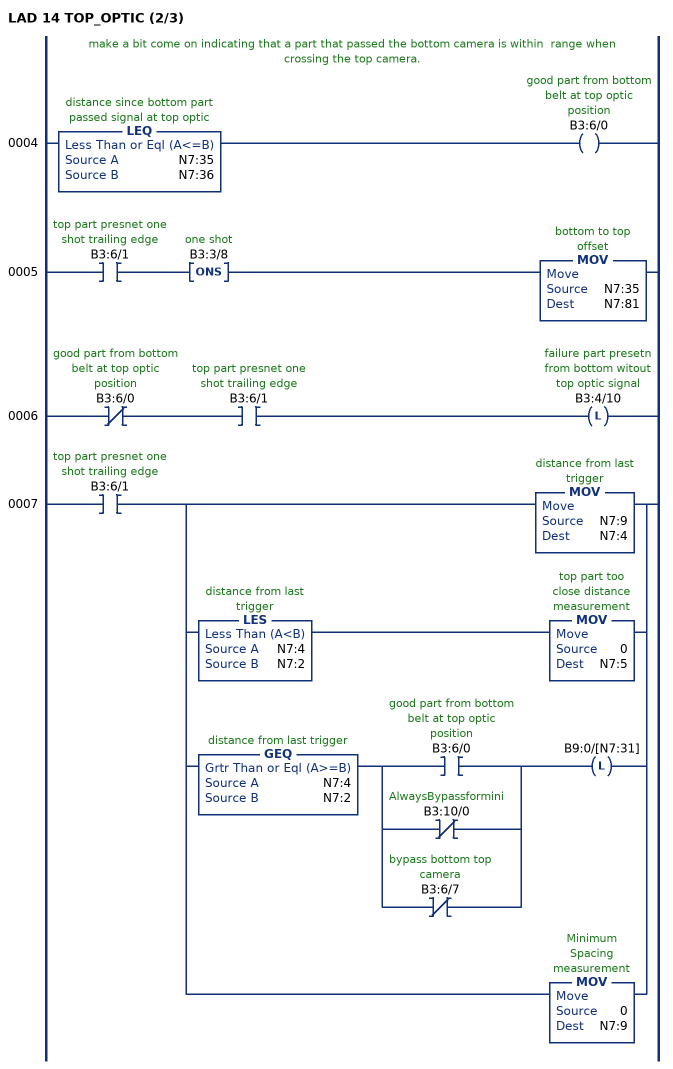
% Rung: 4 %
% make a bit come on indicating that a part that passed the bottom camera is within  range when crossing the top camera. %
SOR LEQ N7:35 N7:36 OTE B3:6/0 EOR
%   N7:35  "distance since bottom part passed signal at top optic" %
%   N7:36  "distance to allow for part shift when part travels from bottom belt to top optic" %
%   B3:6/0  "good part from bottom belt at top optic position" %
% Rung: 5 %
SOR XIC B3:6/1 ONS B3:3/8 MOV N7:35 N7:81 EOR
%   B3:6/1  "top part presnet one shot trailing edge" %
%   B3:3/8  "one shot" %
%   N7:35  "distance since bottom part passed signal at top optic" %
%   N7:81  "bottom to top offset" %
% Rung: 6 %
SOR XIO B3:6/0 XIC B3:6/1 OTL B3:4/10 EOR
%   B3:6/0  "good part from bottom belt at top optic position" %
%   B3:6/1  "top part presnet one shot trailing edge" %
%   B3:4/10  "failure part presetn from bottom witout top optic signal" %
% Rung: 7 %
SOR XIC B3:6/1 BST MOV N7:9 N7:4 NXB LES N7:4 N7:2 MOV 0 N7:5 NXB GEQ N7:4 N7:2 BST XIC B3:6/0 NXB XIO B3:10/0 NXB XIO B3:6/7 BND OTL B9:0/[N7:31] NXB MOV 0 N7:9 BND EOR
%   B3:6/1  "top part presnet one shot trailing edge" %
%   N7:9  "Minimum Spacing measurement" %
%   N7:4  "distance from last trigger" %
%   N7:2  "Min Part Spacing top" %
%   N7:5  "top part too close distance measurement" %
%   B3:6/0  "good part from bottom belt at top optic position" %
%   B3:10/0  "AlwaysBypassformini" %
%   B3:6/7  "bypass bottom top camera" %
%   N7:31  TOP_PART_LOAD_PT %

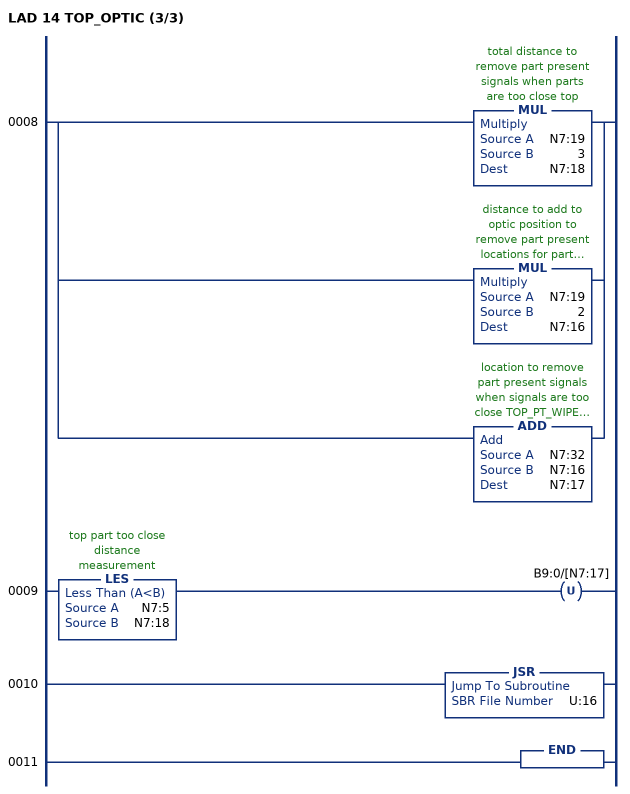
% Rung: 8 %
SOR BST MUL N7:19 3 N7:18 NXB MUL N7:19 2 N7:16 NXB ADD N7:32 N7:16 N7:17 BND EOR
%   N7:19  "distance to remove trigger signals when part spacing too close top" %
%   N7:18  "total distance to remove part present signals when parts are too close top" %
%   N7:16  "distance to add to optic position to remove part present locations for parts too close top" %
%   N7:32  OPTIC_POSITION  "top optic location" %
%   N7:17  TOP_PT_WIPE_LOC  "location to remove part present signals when signals are too close" %
% Rung: 9 %
SOR LES N7:5 N7:18 OTU B9:0/[N7:17] EOR
%   N7:5  "top part too close distance measurement" %
%   N7:18  "total distance to remove part present signals when parts are too close top" %
%   N7:17  TOP_PT_WIPE_LOC  "location to remove part present signals when signals are too close" %
% Rung: 10 %
SOR JSR U:16 EOR
% Rung: 11 %
SOR END EOR

LADDER 16 "TOP_SIDE"
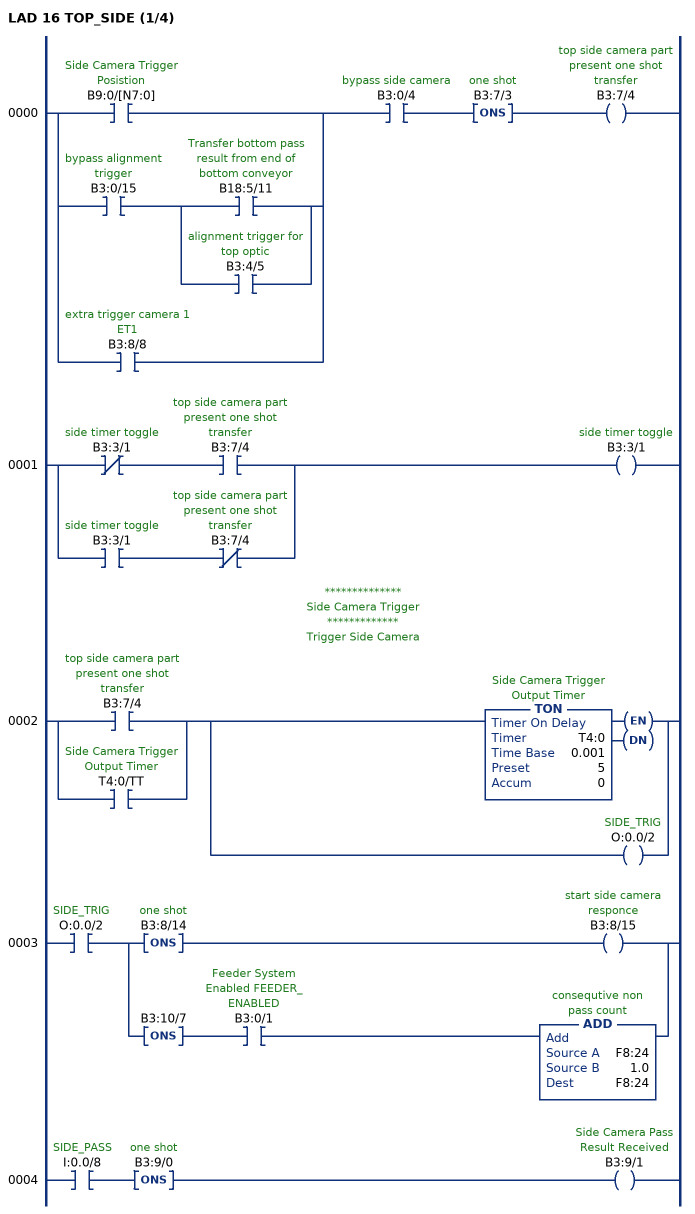
% Rung: 0 %
SOR BST XIC B9:0/[N7:0] NXB XIC B3:0/15 BST XIC B18:5/11 NXB XIC B3:4/5 BND NXB XIC B3:8/8 BND XIC B3:0/4 ONS B3:7/3 OTE B3:7/4 EOR
%   B9:0/[N7:0]  "Side Camera Trigger Posistion" %
%   N7:0  CAMERA_1_SIDE  "Trigger Position" %
%   B3:0/15  "bypass alignment trigger" %
%   B18:5/11  "Transfer bottom pass result from end of bottom conveyor" %
%   B3:4/5  "alignment trigger for top optic" %
%   B3:8/8  ET1  "extra trigger camera 1" %
%   B3:0/4  "bypass side camera" %
%   B3:7/3  "one shot" %
%   B3:7/4  "top side camera part present one shot transfer" %
% Rung: 1 %
SOR BST XIO B3:3/1 XIC B3:7/4 NXB XIC B3:3/1 XIO B3:7/4 BND OTE B3:3/1 EOR
%   B3:3/1  "side timer toggle" %
%   B3:7/4  "top side camera part present one shot transfer" %
% Rung: 2 %
% **************
% Side Camera Trigger
% *************
% 
% Trigger Side Camera %
SOR BST XIC B3:7/4 NXB XIC T4:0/TT BND BST TON T4:0 0.001 5 0 NXB OTE O:0.0/2 BND EOR
%   B3:7/4  "top side camera part present one shot transfer" %
%   T4:0  "Side Camera Trigger Output Timer" %
%   O:0.0/2  SIDE_TRIG %
% Rung: 3 %
SOR XIC O:0.0/2 BST ONS B3:8/14 OTE B3:8/15 NXB ONS B3:10/7 XIC B3:0/1 ADD F8:24 1.0 F8:24 BND EOR
%   O:0.0/2  SIDE_TRIG %
%   B3:8/14  "one shot" %
%   B3:8/15  "start side camera responce" %
%   B3:0/1  FEEDER_ENABLED  "Feeder System Enabled" %
%   F8:24  "consequtive non pass count" %
% Rung: 4 %
SOR XIC I:0.0/8 ONS B3:9/0 OTE B3:9/1 EOR
%   I:0.0/8  SIDE_PASS %
%   B3:9/0  "one shot" %
%   B3:9/1  "Side Camera Pass Result Received" %

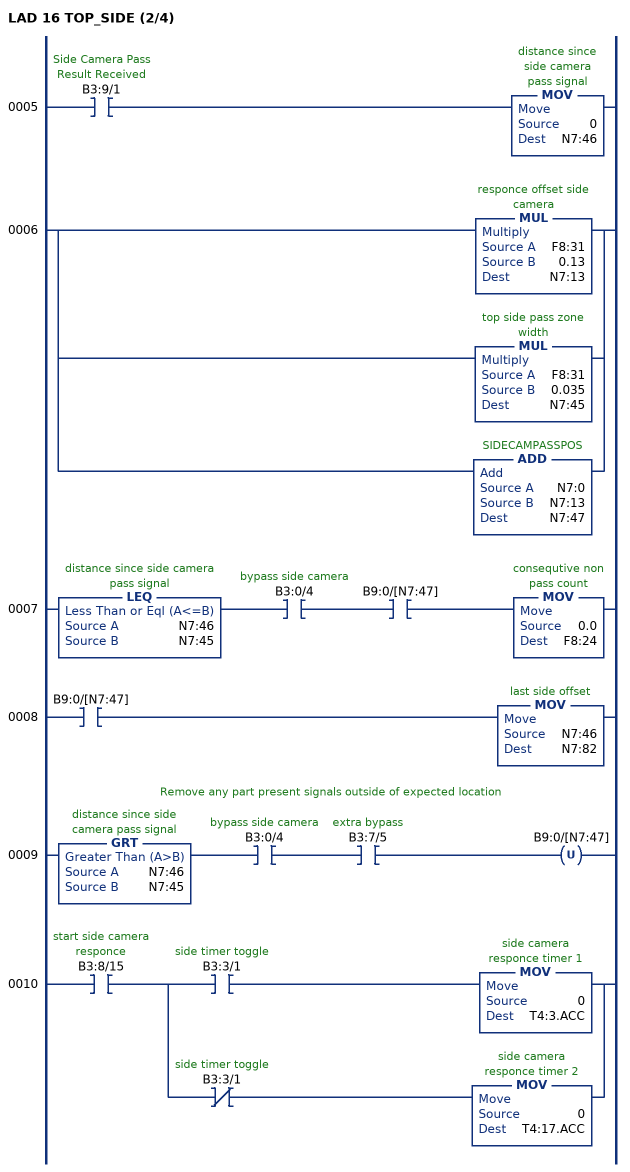
% Rung: 5 %
SOR XIC B3:9/1 MOV 0 N7:46 EOR
%   B3:9/1  "Side Camera Pass Result Received" %
%   N7:46  "distance since side camera pass signal" %
% Rung: 6 %
SOR BST MUL F8:31 0.13 N7:13 NXB MUL F8:31 0.035 N7:45 NXB ADD N7:0 N7:13 N7:47 BND EOR
%   N7:13  "responce offset side camera" %
%   N7:45  "top side pass zone width" %
%   N7:0  CAMERA_1_SIDE  "Trigger Position" %
%   N7:47  SIDECAMPASSPOS %
% Rung: 7 %
SOR LEQ N7:46 N7:45 XIC B3:0/4 XIC B9:0/[N7:47] MOV 0.0 F8:24 EOR
%   N7:46  "distance since side camera pass signal" %
%   N7:45  "top side pass zone width" %
%   B3:0/4  "bypass side camera" %
%   N7:47  SIDECAMPASSPOS %
%   F8:24  "consequtive non pass count" %
% Rung: 8 %
SOR XIC B9:0/[N7:47] MOV N7:46 N7:82 EOR
%   N7:47  SIDECAMPASSPOS %
%   N7:46  "distance since side camera pass signal" %
%   N7:82  "last side offset" %
% Rung: 9 %
% Remove any part present signals outside of expected location %
SOR GRT N7:46 N7:45 XIC B3:0/4 XIC B3:7/5 OTU B9:0/[N7:47] EOR
%   N7:46  "distance since side camera pass signal" %
%   N7:45  "top side pass zone width" %
%   B3:0/4  "bypass side camera" %
%   B3:7/5  "extra bypass" %
%   N7:47  SIDECAMPASSPOS %
% Rung: 10 %
SOR XIC B3:8/15 BST XIC B3:3/1 MOV 0 T4:3.ACC NXB XIO B3:3/1 MOV 0 T4:17.ACC BND EOR
%   B3:8/15  "start side camera responce" %
%   B3:3/1  "side timer toggle" %
%   T4:3  "side camera responce timer 1" %
%   T4:17  "side camera responce timer 2" %

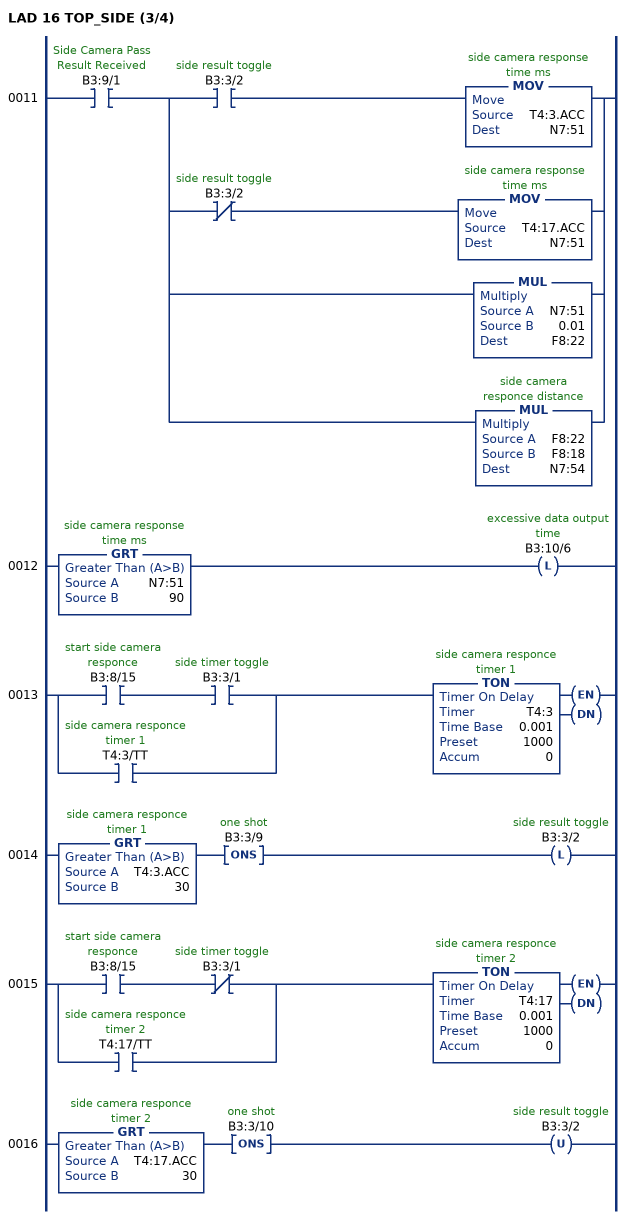
% Rung: 11 %
SOR XIC B3:9/1 BST XIC B3:3/2 MOV T4:3.ACC N7:51 NXB XIO B3:3/2 MOV T4:17.ACC N7:51 NXB MUL N7:51 0.01 F8:22 NXB MUL F8:22 F8:18 N7:54 BND EOR
%   B3:9/1  "Side Camera Pass Result Received" %
%   B3:3/2  "side result toggle" %
%   T4:3  "side camera responce timer 1" %
%   N7:51  "side camera response time ms" %
%   T4:17  "side camera responce timer 2" %
%   F8:18  "top belt speed average in pulses per 100ms" %
%   N7:54  "side camera responce distance" %
% Rung: 12 %
SOR GRT N7:51 90 OTL B3:10/6 EOR
%   N7:51  "side camera response time ms" %
%   B3:10/6  "excessive data output time" %
% Rung: 13 %
SOR BST XIC B3:8/15 XIC B3:3/1 NXB XIC T4:3/TT BND TON T4:3 0.001 1000 0 EOR
%   B3:8/15  "start side camera responce" %
%   B3:3/1  "side timer toggle" %
%   T4:3  "side camera responce timer 1" %
% Rung: 14 %
SOR GRT T4:3.ACC 30 ONS B3:3/9 OTL B3:3/2 EOR
%   T4:3  "side camera responce timer 1" %
%   B3:3/9  "one shot" %
%   B3:3/2  "side result toggle" %
% Rung: 15 %
SOR BST XIC B3:8/15 XIO B3:3/1 NXB XIC T4:17/TT BND TON T4:17 0.001 1000 0 EOR
%   B3:8/15  "start side camera responce" %
%   B3:3/1  "side timer toggle" %
%   T4:17  "side camera responce timer 2" %
% Rung: 16 %
SOR GRT T4:17.ACC 30 ONS B3:3/10 OTU B3:3/2 EOR
%   T4:17  "side camera responce timer 2" %
%   B3:3/10  "one shot" %
%   B3:3/2  "side result toggle" %

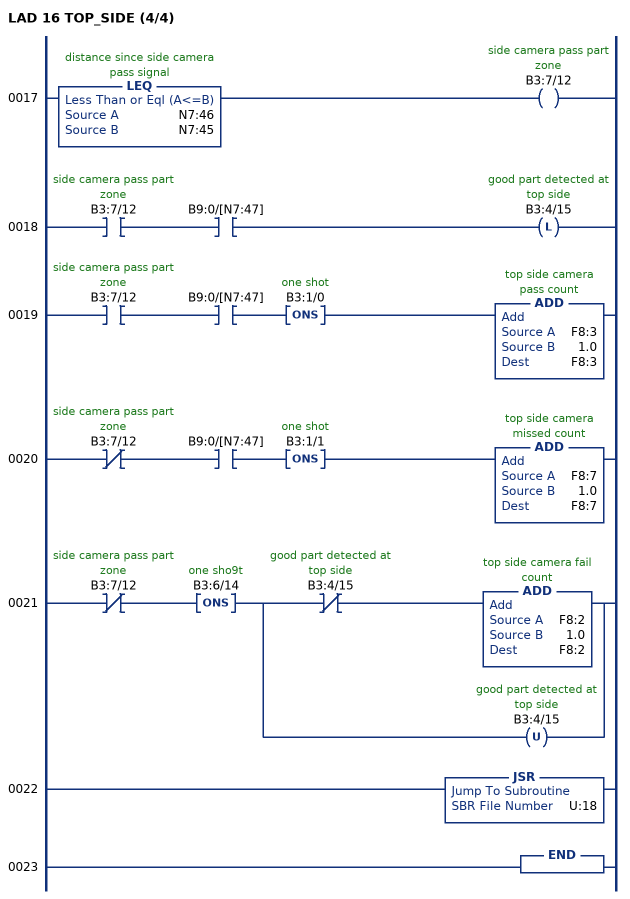
% Rung: 17 %
SOR LEQ N7:46 N7:45 OTE B3:7/12 EOR
%   N7:46  "distance since side camera pass signal" %
%   N7:45  "top side pass zone width" %
%   B3:7/12  "side camera pass part zone" %
% Rung: 18 %
SOR XIC B3:7/12 XIC B9:0/[N7:47] OTL B3:4/15 EOR
%   B3:7/12  "side camera pass part zone" %
%   N7:47  SIDECAMPASSPOS %
%   B3:4/15  "good part detected at top side" %
% Rung: 19 %
SOR XIC B3:7/12 XIC B9:0/[N7:47] ONS B3:1/0 ADD F8:3 1.0 F8:3 EOR
%   B3:7/12  "side camera pass part zone" %
%   N7:47  SIDECAMPASSPOS %
%   B3:1/0  "one shot" %
%   F8:3  "top side camera pass count" %
% Rung: 20 %
SOR XIO B3:7/12 XIC B9:0/[N7:47] ONS B3:1/1 ADD F8:7 1.0 F8:7 EOR
%   B3:7/12  "side camera pass part zone" %
%   N7:47  SIDECAMPASSPOS %
%   B3:1/1  "one shot" %
%   F8:7  "top side camera missed count" %
% Rung: 21 %
SOR XIO B3:7/12 ONS B3:6/14 BST XIO B3:4/15 ADD F8:2 1.0 F8:2 NXB OTU B3:4/15 BND EOR
%   B3:7/12  "side camera pass part zone" %
%   B3:6/14  "one sho9t" %
%   B3:4/15  "good part detected at top side" %
%   F8:2  "top side camera fail count" %
% Rung: 22 %
SOR JSR U:18 EOR
% Rung: 23 %
SOR END EOR

LADDER 18 "TOP_PYRIMI"
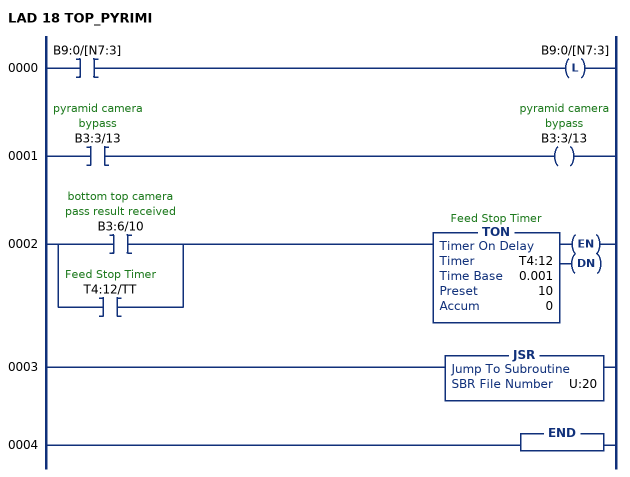
% Rung: 0 %
SOR XIC B9:0/[N7:3] OTL B9:0/[N7:3] EOR
%   N7:3  PYRAMID_TRIG  "pyramid camera trigger position" %
% Rung: 1 %
SOR XIC B3:3/13 OTE B3:3/13 EOR
%   B3:3/13  "pyramid camera bypass" %
% Rung: 2 %
SOR BST XIC B3:6/10 NXB XIC T4:12/TT BND TON T4:12 0.001 10 0 EOR
%   B3:6/10  "bottom top camera pass result received" %
%   T4:12  "Feed Stop Timer" %
% Rung: 3 %
SOR JSR U:20 EOR
% Rung: 4 %
SOR END EOR

LADDER 20 "TOP_TOP"
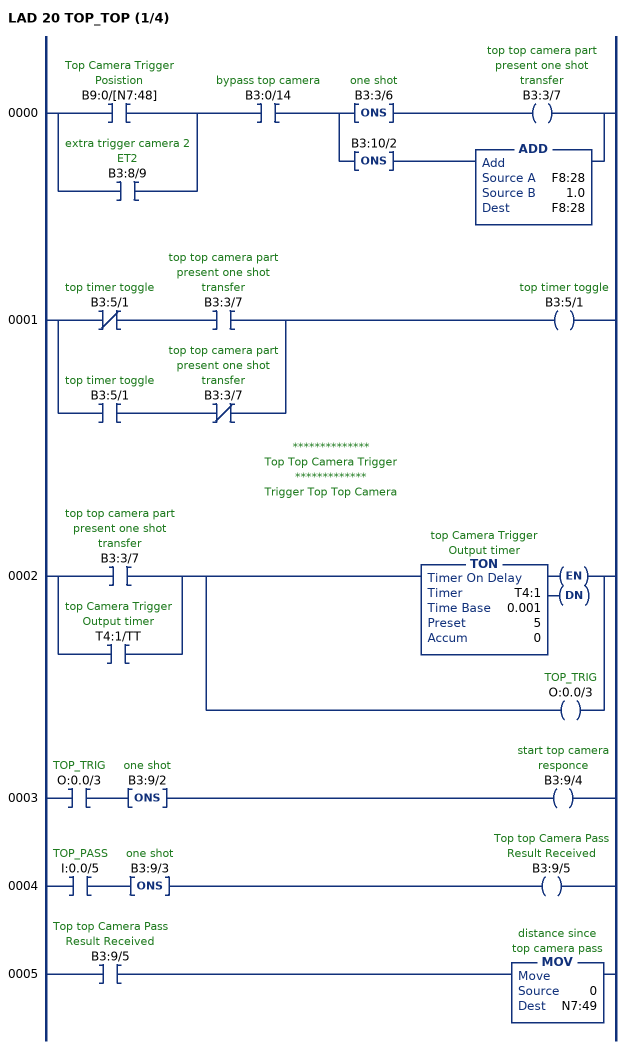
% Rung: 0 %
SOR BST XIC B9:0/[N7:48] NXB XIC B3:8/9 BND XIC B3:0/14 BST ONS B3:3/6 OTE B3:3/7 NXB ONS B3:10/2 ADD F8:28 1.0 F8:28 BND EOR
%   B9:0/[N7:48]  "Top Camera Trigger Posistion" %
%   N7:48  CAMERA_2_TOP  "top camera trigger position" %
%   B3:8/9  ET2  "extra trigger camera 2" %
%   B3:0/14  "bypass top camera" %
%   B3:3/6  "one shot" %
%   B3:3/7  "top top camera part present one shot transfer" %
% Rung: 1 %
SOR BST XIO B3:5/1 XIC B3:3/7 NXB XIC B3:5/1 XIO B3:3/7 BND OTE B3:5/1 EOR
%   B3:5/1  "top timer toggle" %
%   B3:3/7  "top top camera part present one shot transfer" %
% Rung: 2 %
% **************
% Top Top Camera Trigger
% *************
% 
% Trigger Top Top Camera %
SOR BST XIC B3:3/7 NXB XIC T4:1/TT BND BST TON T4:1 0.001 5 0 NXB OTE O:0.0/3 BND EOR
%   B3:3/7  "top top camera part present one shot transfer" %
%   T4:1  "top Camera Trigger Output timer" %
%   O:0.0/3  TOP_TRIG %
% Rung: 3 %
SOR XIC O:0.0/3 ONS B3:9/2 OTE B3:9/4 EOR
%   O:0.0/3  TOP_TRIG %
%   B3:9/2  "one shot" %
%   B3:9/4  "start top camera responce" %
% Rung: 4 %
SOR XIC I:0.0/5 ONS B3:9/3 OTE B3:9/5 EOR
%   I:0.0/5  TOP_PASS %
%   B3:9/3  "one shot" %
%   B3:9/5  "Top top Camera Pass Result Received" %
% Rung: 5 %
SOR XIC B3:9/5 MOV 0 N7:49 EOR
%   B3:9/5  "Top top Camera Pass Result Received" %
%   N7:49  "distance since top camera pass" %

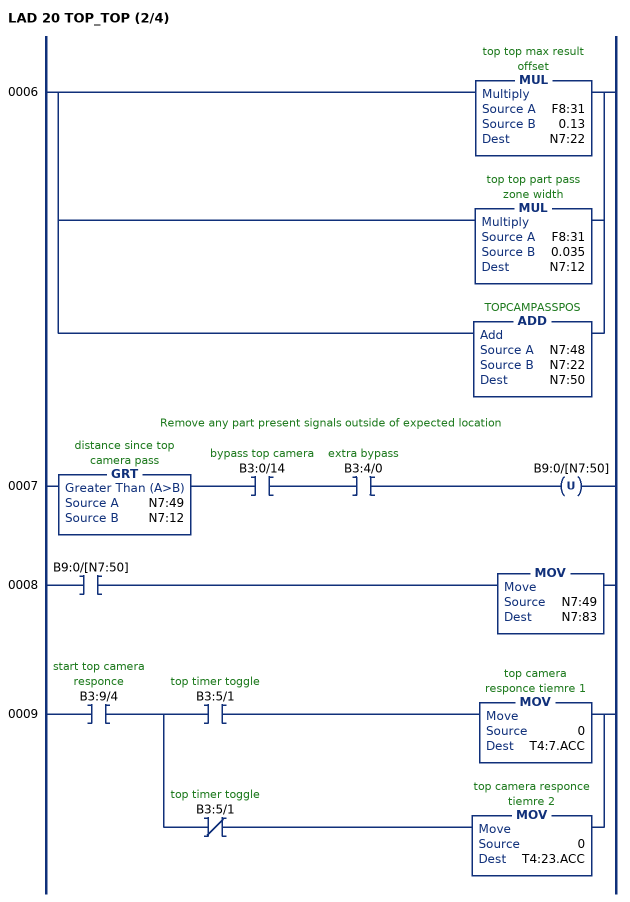
% Rung: 6 %
SOR BST MUL F8:31 0.13 N7:22 NXB MUL F8:31 0.035 N7:12 NXB ADD N7:48 N7:22 N7:50 BND EOR
%   N7:22  "top top max result offset" %
%   N7:12  "top top part pass zone width" %
%   N7:48  CAMERA_2_TOP  "top camera trigger position" %
%   N7:50  TOPCAMPASSPOS %
% Rung: 7 %
% Remove any part present signals outside of expected location %
SOR GRT N7:49 N7:12 XIC B3:0/14 XIC B3:4/0 OTU B9:0/[N7:50] EOR
%   N7:49  "distance since top camera pass" %
%   N7:12  "top top part pass zone width" %
%   B3:0/14  "bypass top camera" %
%   B3:4/0  "extra bypass" %
%   N7:50  TOPCAMPASSPOS %
% Rung: 8 %
SOR XIC B9:0/[N7:50] MOV N7:49 N7:83 EOR
%   N7:50  TOPCAMPASSPOS %
%   N7:49  "distance since top camera pass" %
% Rung: 9 %
SOR XIC B3:9/4 BST XIC B3:5/1 MOV 0 T4:7.ACC NXB XIO B3:5/1 MOV 0 T4:23.ACC BND EOR
%   B3:9/4  "start top camera responce" %
%   B3:5/1  "top timer toggle" %
%   T4:7  "top camera responce tiemre 1" %
%   T4:23  "top camera responce tiemre 2" %

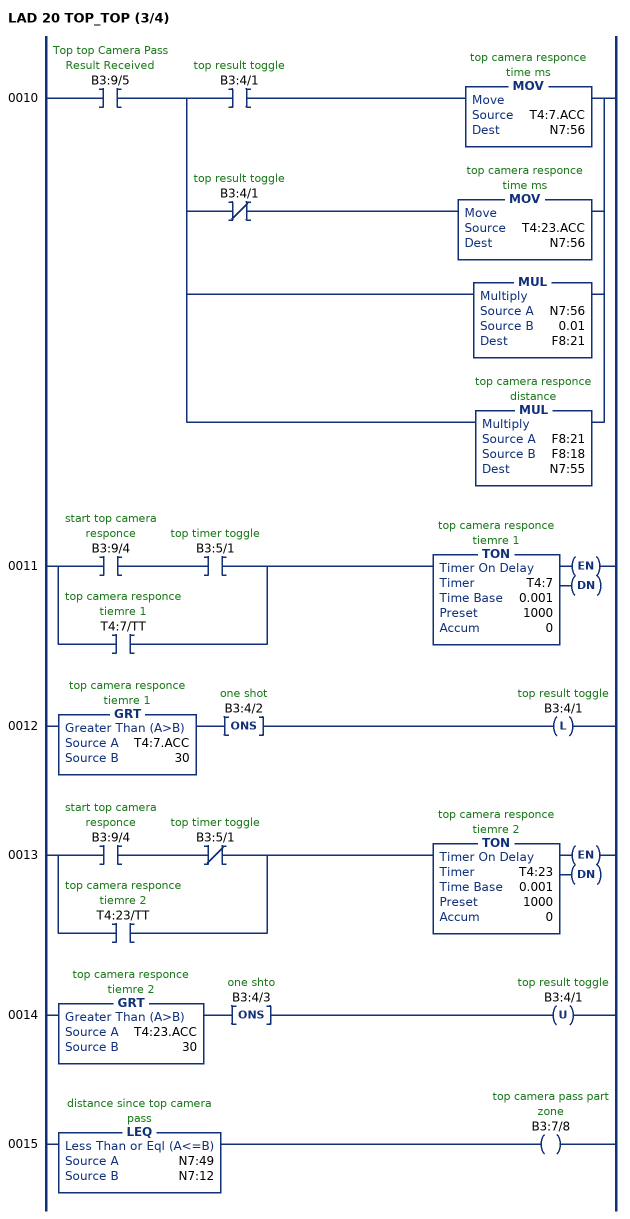
% Rung: 10 %
SOR XIC B3:9/5 BST XIC B3:4/1 MOV T4:7.ACC N7:56 NXB XIO B3:4/1 MOV T4:23.ACC N7:56 NXB MUL N7:56 0.01 F8:21 NXB MUL F8:21 F8:18 N7:55 BND EOR
%   B3:9/5  "Top top Camera Pass Result Received" %
%   B3:4/1  "top result toggle" %
%   T4:7  "top camera responce tiemre 1" %
%   N7:56  "top camera responce time ms" %
%   T4:23  "top camera responce tiemre 2" %
%   F8:18  "top belt speed average in pulses per 100ms" %
%   N7:55  "top camera responce distance" %
% Rung: 11 %
SOR BST XIC B3:9/4 XIC B3:5/1 NXB XIC T4:7/TT BND TON T4:7 0.001 1000 0 EOR
%   B3:9/4  "start top camera responce" %
%   B3:5/1  "top timer toggle" %
%   T4:7  "top camera responce tiemre 1" %
% Rung: 12 %
SOR GRT T4:7.ACC 30 ONS B3:4/2 OTL B3:4/1 EOR
%   T4:7  "top camera responce tiemre 1" %
%   B3:4/2  "one shot" %
%   B3:4/1  "top result toggle" %
% Rung: 13 %
SOR BST XIC B3:9/4 XIO B3:5/1 NXB XIC T4:23/TT BND TON T4:23 0.001 1000 0 EOR
%   B3:9/4  "start top camera responce" %
%   B3:5/1  "top timer toggle" %
%   T4:23  "top camera responce tiemre 2" %
% Rung: 14 %
SOR GRT T4:23.ACC 30 ONS B3:4/3 OTU B3:4/1 EOR
%   T4:23  "top camera responce tiemre 2" %
%   B3:4/3  "one shto" %
%   B3:4/1  "top result toggle" %
% Rung: 15 %
SOR LEQ N7:49 N7:12 OTE B3:7/8 EOR
%   N7:49  "distance since top camera pass" %
%   N7:12  "top top part pass zone width" %
%   B3:7/8  "top camera pass part zone" %

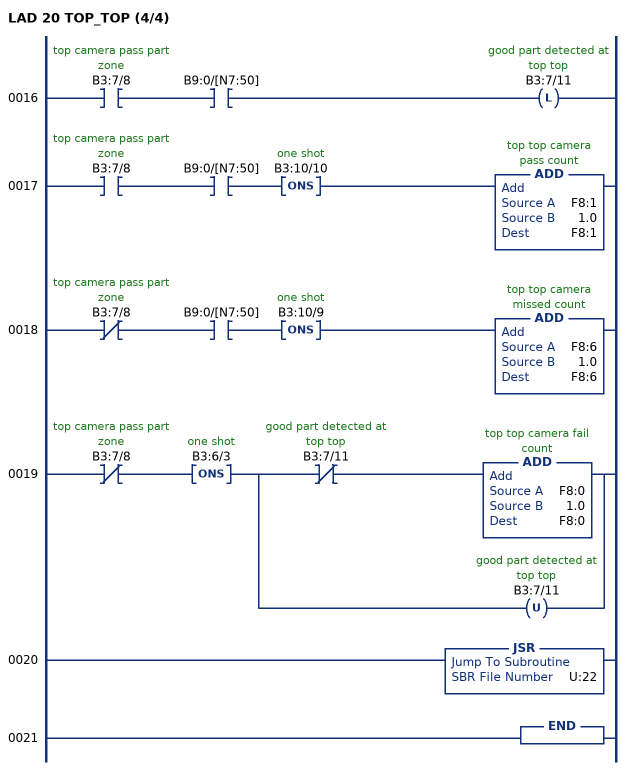
% Rung: 16 %
SOR XIC B3:7/8 XIC B9:0/[N7:50] OTL B3:7/11 EOR
%   B3:7/8  "top camera pass part zone" %
%   N7:50  TOPCAMPASSPOS %
%   B3:7/11  "good part detected at top top" %
% Rung: 17 %
SOR XIC B3:7/8 XIC B9:0/[N7:50] ONS B3:10/10 ADD F8:1 1.0 F8:1 EOR
%   B3:7/8  "top camera pass part zone" %
%   N7:50  TOPCAMPASSPOS %
%   B3:10/10  "one shot" %
%   F8:1  "top top camera pass count" %
% Rung: 18 %
SOR XIO B3:7/8 XIC B9:0/[N7:50] ONS B3:10/9 ADD F8:6 1.0 F8:6 EOR
%   B3:7/8  "top camera pass part zone" %
%   N7:50  TOPCAMPASSPOS %
%   B3:10/9  "one shot" %
%   F8:6  "top top camera missed count" %
% Rung: 19 %
SOR XIO B3:7/8 ONS B3:6/3 BST XIO B3:7/11 ADD F8:0 1.0 F8:0 NXB OTU B3:7/11 BND EOR
%   B3:7/8  "top camera pass part zone" %
%   B3:6/3  "one shot" %
%   B3:7/11  "good part detected at top top" %
%   F8:0  "top top camera fail count" %
% Rung: 20 %
SOR JSR U:22 EOR
% Rung: 21 %
SOR END EOR

LADDER 22 "TOP_THREAD"
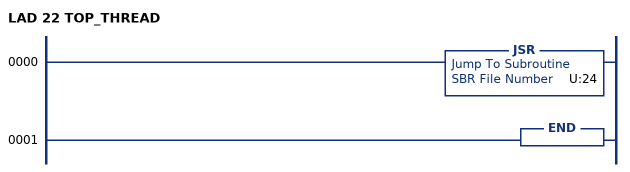
% Rung: 0 %
SOR JSR U:24 EOR
% Rung: 1 %
SOR END EOR

LADDER 24 "TOP_BLOW"
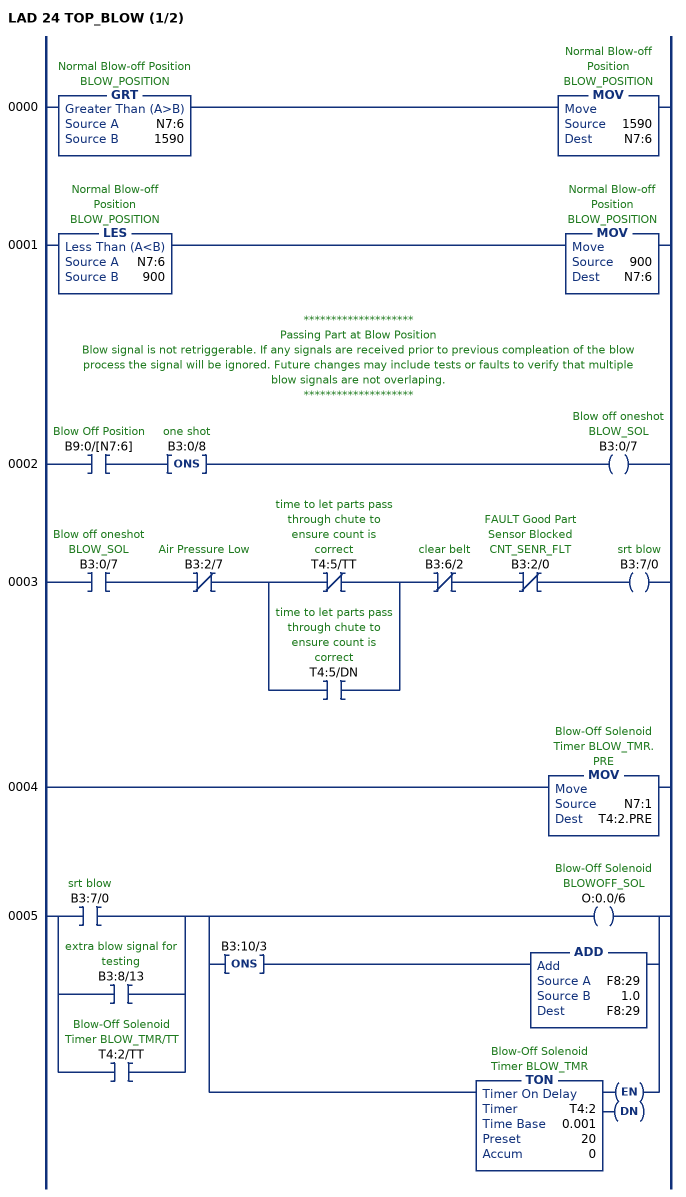
% Rung: 0 %
SOR GRT N7:6 1590 MOV 1590 N7:6 EOR
%   N7:6  BLOW_POSITION  "Normal Blow-off Position" %
% Rung: 1 %
SOR LES N7:6 900 MOV 900 N7:6 EOR
%   N7:6  BLOW_POSITION  "Normal Blow-off Position" %
% Rung: 2 %
% ********************
% Passing Part at Blow Position
% 
% Blow signal is not retriggerable. If any signals are received prior to previous compleation of the blow process the signal will be ignored. Future changes may include tests or faults to verify that multiple blow signals are not overlaping.
% ******************** %
SOR XIC B9:0/[N7:6] ONS B3:0/8 OTE B3:0/7 EOR
%   B9:0/[N7:6]  "Blow Off Position" %
%   N7:6  BLOW_POSITION  "Normal Blow-off Position" %
%   B3:0/8  "one shot" %
%   B3:0/7  BLOW_SOL  "Blow off oneshot" %
% Rung: 3 %
SOR XIC B3:0/7 XIO B3:2/7 BST XIO T4:5/TT NXB XIC T4:5/DN BND XIO B3:6/2 XIO B3:2/0 OTE B3:7/0 EOR
%   B3:0/7  BLOW_SOL  "Blow off oneshot" %
%   B3:2/7  "Air Pressure Low" %
%   T4:5  "time to let parts pass through chute to ensure count is correct" %
%   B3:6/2  "clear belt" %
%   B3:2/0  CNT_SENR_FLT  "FAULT Good Part Sensor Blocked" %
%   B3:7/0  "srt blow" %
% Rung: 4 %
SOR MOV N7:1 T4:2.PRE EOR
%   N7:1  "Blow off Time" %
%   T4:2  BLOW_TMR  "Blow-Off Solenoid Timer" %
% Rung: 5 %
SOR BST XIC B3:7/0 NXB XIC B3:8/13 NXB XIC T4:2/TT BND BST OTE O:0.0/6 NXB ONS B3:10/3 ADD F8:29 1.0 F8:29 NXB TON T4:2 0.001 20 0 BND EOR
%   B3:7/0  "srt blow" %
%   B3:8/13  "extra blow signal for testing" %
%   T4:2  BLOW_TMR  "Blow-Off Solenoid Timer" %
%   O:0.0/6  BLOWOFF_SOL  "Blow-Off Solenoid" %

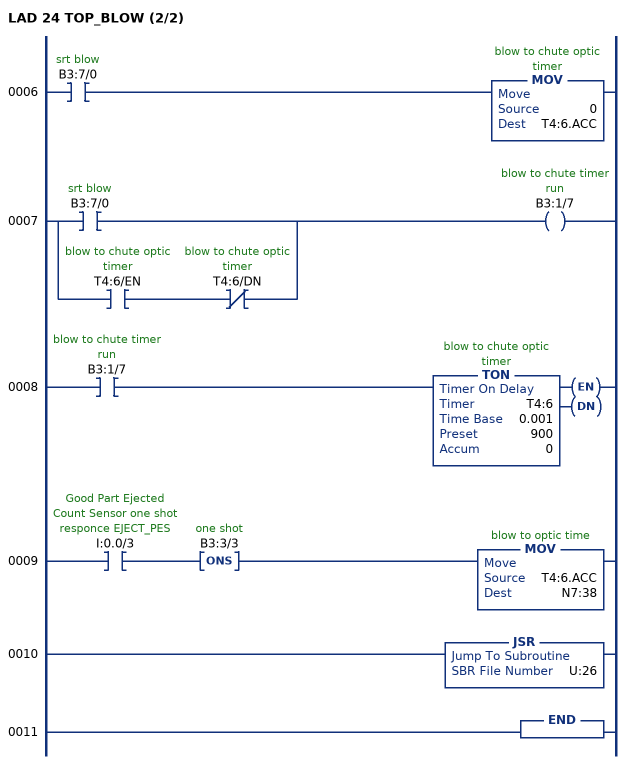
% Rung: 6 %
SOR XIC B3:7/0 MOV 0 T4:6.ACC EOR
%   B3:7/0  "srt blow" %
%   T4:6  "blow to chute optic timer" %
% Rung: 7 %
SOR BST XIC B3:7/0 NXB XIC T4:6/EN XIO T4:6/DN BND OTE B3:1/7 EOR
%   B3:7/0  "srt blow" %
%   T4:6  "blow to chute optic timer" %
%   B3:1/7  "blow to chute timer run" %
% Rung: 8 %
SOR XIC B3:1/7 TON T4:6 0.001 900 0 EOR
%   B3:1/7  "blow to chute timer run" %
%   T4:6  "blow to chute optic timer" %
% Rung: 9 %
SOR XIC I:0.0/3 ONS B3:3/3 MOV T4:6.ACC N7:38 EOR
%   I:0.0/3  EJECT_PES  "Good Part Ejected Count Sensor one shot responce" %
%   B3:3/3  "one shot" %
%   T4:6  "blow to chute optic timer" %
%   N7:38  "blow to optic time" %
% Rung: 10 %
SOR JSR U:26 EOR
% Rung: 11 %
SOR END EOR

LADDER 26 "FLOW"
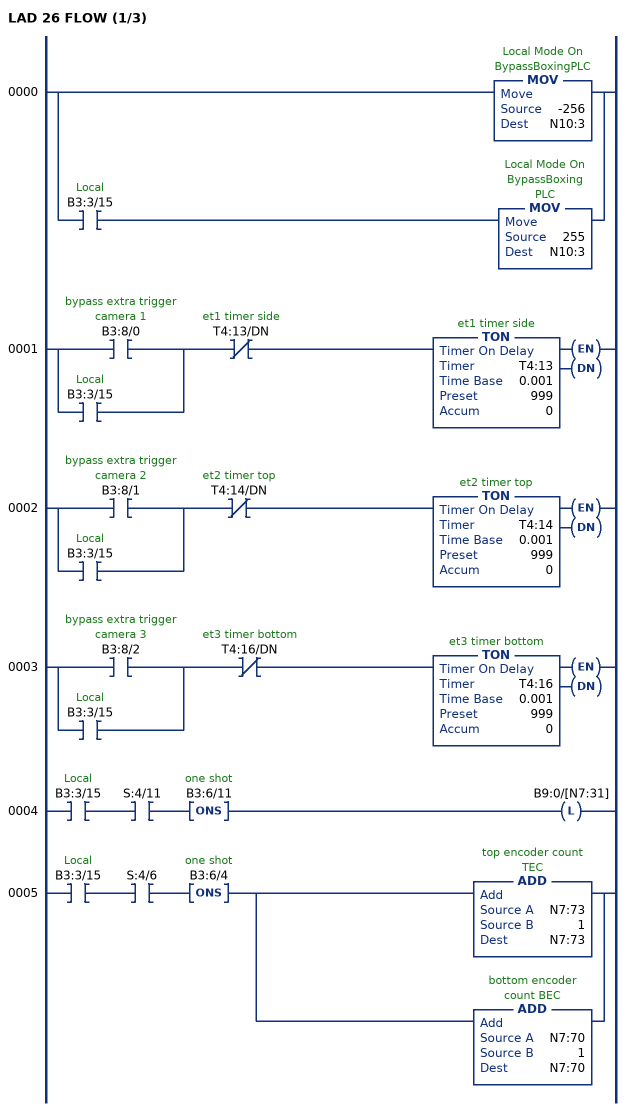
% Rung: 0 %
SOR BST MOV -256 N10:3 NXB XIC B3:3/15 MOV 255 N10:3 BND EOR
%   N10:3  "Local Mode On BypassBoxingPLC" %
%   B3:3/15  "Local" %
% Rung: 1 %
SOR BST XIC B3:8/0 NXB XIC B3:3/15 BND XIO T4:13/DN TON T4:13 0.001 999 0 EOR
%   B3:8/0  "bypass extra trigger camera 1" %
%   B3:3/15  "Local" %
%   T4:13  "et1 timer side" %
% Rung: 2 %
SOR BST XIC B3:8/1 NXB XIC B3:3/15 BND XIO T4:14/DN TON T4:14 0.001 999 0 EOR
%   B3:8/1  "bypass extra trigger camera 2" %
%   B3:3/15  "Local" %
%   T4:14  "et2 timer top" %
% Rung: 3 %
SOR BST XIC B3:8/2 NXB XIC B3:3/15 BND XIO T4:16/DN TON T4:16 0.001 999 0 EOR
%   B3:8/2  "bypass extra trigger camera 3" %
%   B3:3/15  "Local" %
%   T4:16  "et3 timer bottom" %
% Rung: 4 %
SOR XIC B3:3/15 XIC S:4/11 ONS B3:6/11 OTL B9:0/[N7:31] EOR
%   B3:3/15  "Local" %
%   B3:6/11  "one shot" %
%   N7:31  TOP_PART_LOAD_PT %
% Rung: 5 %
SOR XIC B3:3/15 XIC S:4/6 ONS B3:6/4 BST ADD N7:73 1 N7:73 NXB ADD N7:70 1 N7:70 BND EOR
%   B3:3/15  "Local" %
%   B3:6/4  "one shot" %
%   N7:73  TEC  "top encoder count" %
%   N7:70  BEC  "bottom encoder count" %

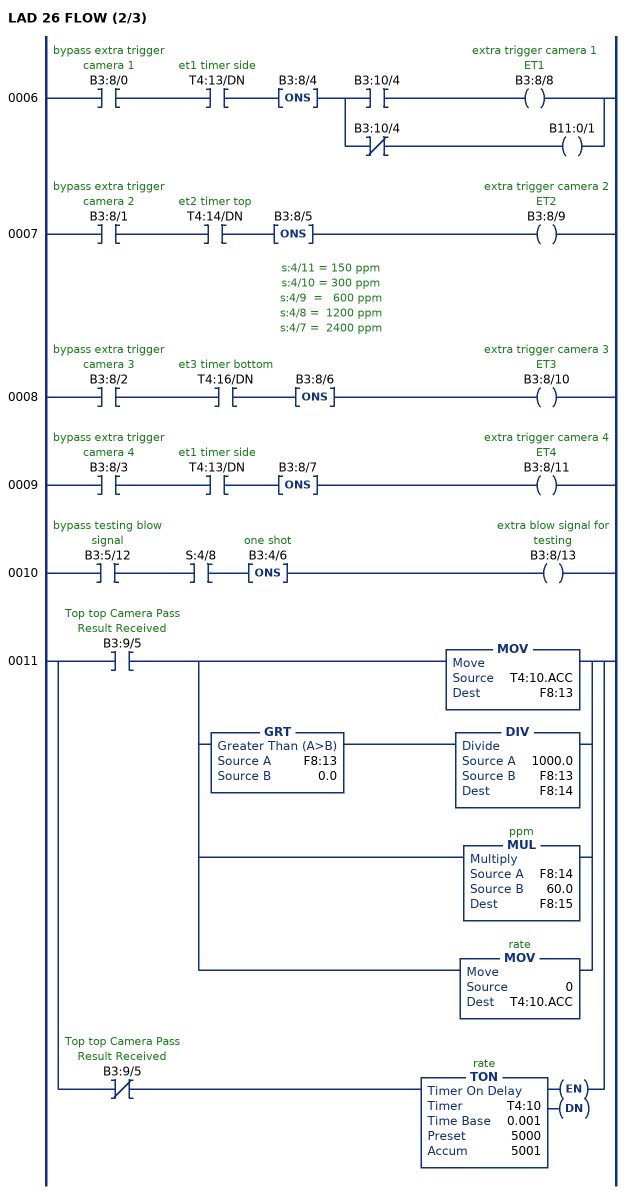
% Rung: 6 %
SOR XIC B3:8/0 XIC T4:13/DN ONS B3:8/4 BST XIC B3:10/4 OTE B3:8/8 NXB XIO B3:10/4 OTE B11:0/1 BND EOR
%   B3:8/0  "bypass extra trigger camera 1" %
%   T4:13  "et1 timer side" %
%   B3:8/8  ET1  "extra trigger camera 1" %
% Rung: 7 %
SOR XIC B3:8/1 XIC T4:14/DN ONS B3:8/5 OTE B3:8/9 EOR
%   B3:8/1  "bypass extra trigger camera 2" %
%   T4:14  "et2 timer top" %
%   B3:8/9  ET2  "extra trigger camera 2" %
% Rung: 8 %
% s:4/11 = 150 ppm
% s:4/10 = 300 ppm
% s:4/9  =   600 ppm
% s:4/8 =  1200 ppm
% s:4/7 =  2400 ppm %
SOR XIC B3:8/2 XIC T4:16/DN ONS B3:8/6 OTE B3:8/10 EOR
%   B3:8/2  "bypass extra trigger camera 3" %
%   T4:16  "et3 timer bottom" %
%   B3:8/10  ET3  "extra trigger camera 3" %
% Rung: 9 %
SOR XIC B3:8/3 XIC T4:13/DN ONS B3:8/7 OTE B3:8/11 EOR
%   B3:8/3  "bypass extra trigger camera 4" %
%   T4:13  "et1 timer side" %
%   B3:8/11  ET4  "extra trigger camera 4" %
% Rung: 10 %
SOR XIC B3:5/12 XIC S:4/8 ONS B3:4/6 OTE B3:8/13 EOR
%   B3:5/12  "bypass testing blow signal" %
%   B3:4/6  "one shot" %
%   B3:8/13  "extra blow signal for testing" %
% Rung: 11 %
SOR BST XIC B3:9/5 BST MOV T4:10.ACC F8:13 NXB GRT F8:13 0.0 DIV 1000.0 F8:13 F8:14 NXB MUL F8:14 60.0 F8:15 NXB MOV 0 T4:10.ACC BND NXB XIO B3:9/5 TON T4:10 0.001 5000 5001 BND EOR
%   B3:9/5  "Top top Camera Pass Result Received" %
%   T4:10  "rate" %
%   F8:15  "ppm" %

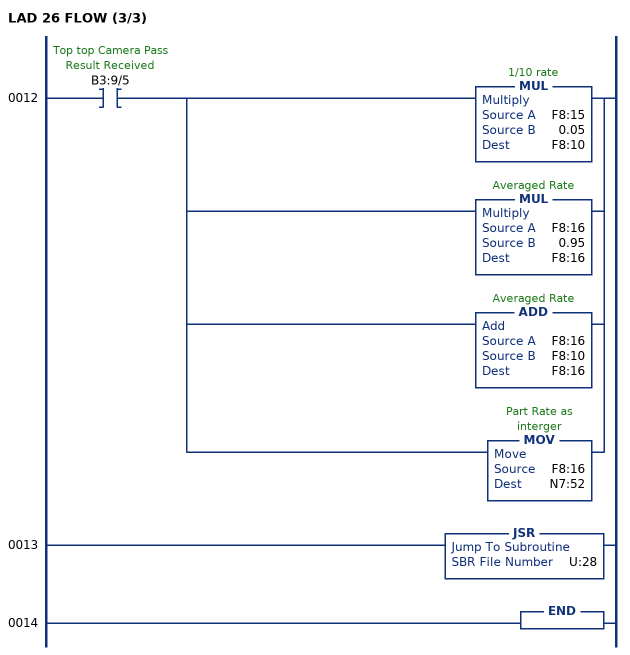
% Rung: 12 %
SOR XIC B3:9/5 BST MUL F8:15 0.05 F8:10 NXB MUL F8:16 0.95 F8:16 NXB ADD F8:16 F8:10 F8:16 NXB MOV F8:16 N7:52 BND EOR
%   B3:9/5  "Top top Camera Pass Result Received" %
%   F8:15  "ppm" %
%   F8:10  "1/10 rate" %
%   F8:16  "Averaged Rate" %
%   N7:52  "Part Rate as interger" %
% Rung: 13 %
SOR JSR U:28 EOR
% Rung: 14 %
SOR END EOR

LADDER 28 "FAULTS"
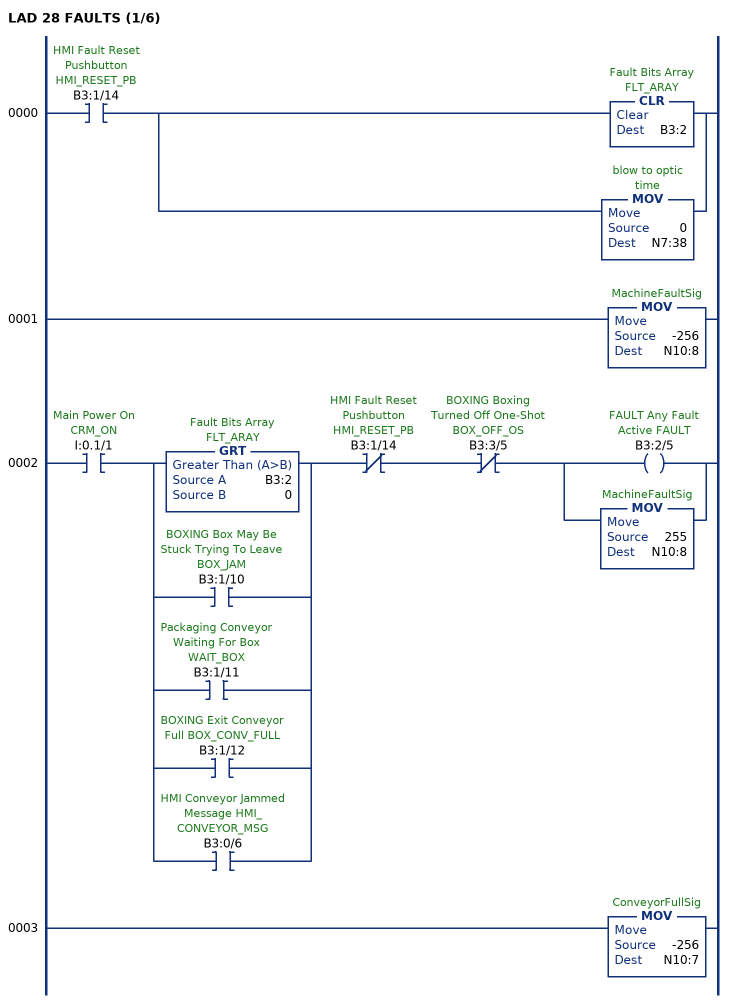
% Rung: 0 %
SOR XIC B3:1/14 BST CLR B3:2 NXB MOV 0 N7:38 BND EOR
%   B3:1/14  HMI_RESET_PB  "HMI Fault Reset Pushbutton" %
%   B3:2  FLT_ARAY  "Fault Bits Array" %
%   N7:38  "blow to optic time" %
% Rung: 1 %
SOR MOV -256 N10:8 EOR
%   N10:8  "MachineFaultSig" %
% Rung: 2 %
SOR XIC I:0.1/1 BST GRT B3:2 0 NXB XIC B3:1/10 NXB XIC B3:1/11 NXB XIC B3:1/12 NXB XIC B3:0/6 BND XIO B3:1/14 XIO B3:3/5 BST OTE B3:2/5 NXB MOV 255 N10:8 BND EOR
%   I:0.1/1  CRM_ON  "Main Power On" %
%   B3:2  FLT_ARAY  "Fault Bits Array" %
%   B3:1/10  BOX_JAM  "BOXING Box May Be Stuck Trying To Leave" %
%   B3:1/11  WAIT_BOX  "Packaging Conveyor Waiting For Box" %
%   B3:1/12  BOX_CONV_FULL  "BOXING Exit Conveyor Full" %
%   B3:0/6  HMI_CONVEYOR_MSG  "HMI Conveyor Jammed Message" %
%   B3:1/14  HMI_RESET_PB  "HMI Fault Reset Pushbutton" %
%   B3:3/5  BOX_OFF_OS  "BOXING Boxing Turned Off One-Shot" %
%   B3:2/5  FAULT  "FAULT Any Fault Active" %
%   N10:8  "MachineFaultSig" %
% Rung: 3 %
SOR MOV -256 N10:7 EOR
%   N10:7  "ConveyorFullSig" %

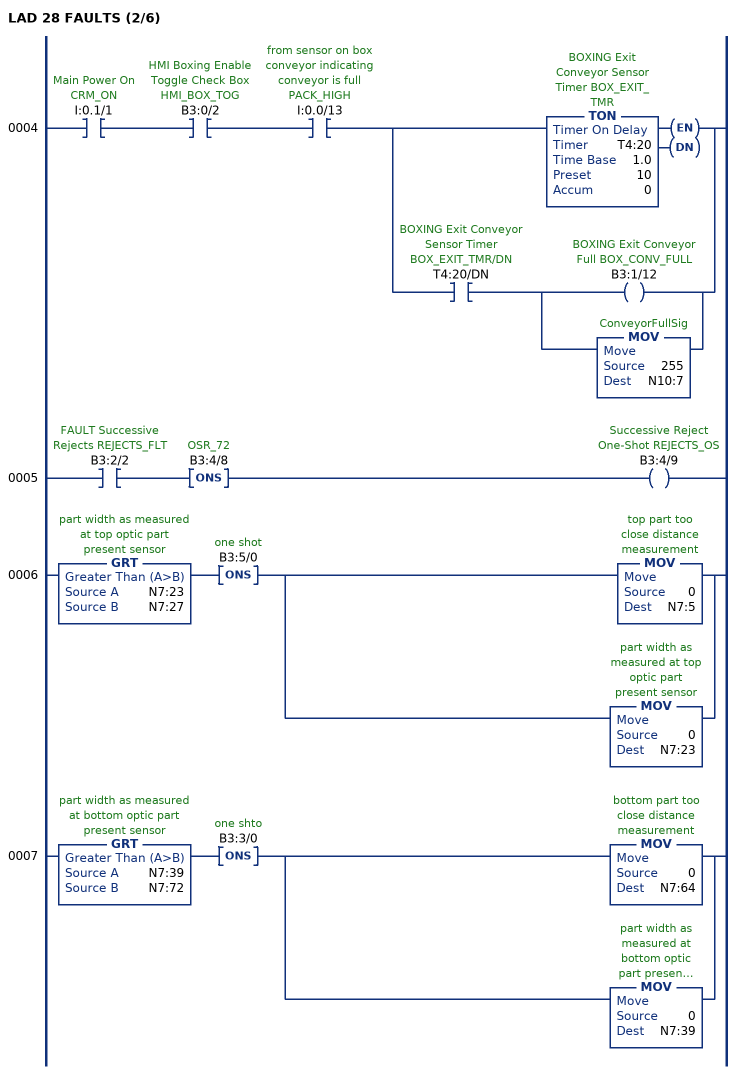
% Rung: 4 %
SOR XIC I:0.1/1 XIC B3:0/2 XIC I:0.0/13 BST TON T4:20 1.0 10 0 NXB XIC T4:20/DN BST OTE B3:1/12 NXB MOV 255 N10:7 BND BND EOR
%   I:0.1/1  CRM_ON  "Main Power On" %
%   B3:0/2  HMI_BOX_TOG  "HMI Boxing Enable Toggle Check Box" %
%   I:0.0/13  PACK_HIGH  "from sensor on box conveyor indicating conveyor is full" %
%   T4:20  BOX_EXIT_TMR  "BOXING Exit Conveyor Sensor Timer" %
%   B3:1/12  BOX_CONV_FULL  "BOXING Exit Conveyor Full" %
%   N10:7  "ConveyorFullSig" %
% Rung: 5 %
SOR XIC B3:2/2 ONS B3:4/8 OTE B3:4/9 EOR
%   B3:2/2  REJECTS_FLT  "FAULT Successive Rejects" %
%   B3:4/8  OSR_72 %
%   B3:4/9  REJECTS_OS  "Successive Reject One-Shot" %
% Rung: 6 %
SOR GRT N7:23 N7:27 ONS B3:5/0 BST MOV 0 N7:5 NXB MOV 0 N7:23 BND EOR
%   N7:23  "part width as measured at top optic part present sensor" %
%   N7:27  "max part width top optic" %
%   B3:5/0  "one shot" %
%   N7:5  "top part too close distance measurement" %
% Rung: 7 %
SOR GRT N7:39 N7:72 ONS B3:3/0 BST MOV 0 N7:64 NXB MOV 0 N7:39 BND EOR
%   N7:39  "part width as measured at bottom optic part present sensor" %
%   N7:72  "max part width bottom optic" %
%   B3:3/0  "one shto" %
%   N7:64  "bottom part too close distance measurement" %

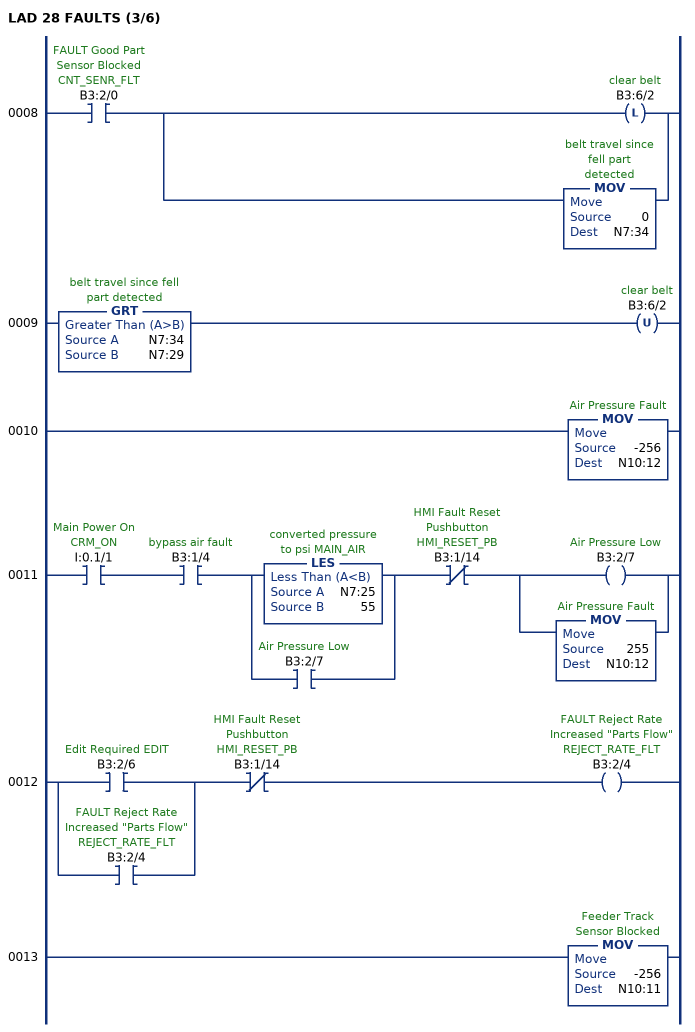
% Rung: 8 %
SOR XIC B3:2/0 BST OTL B3:6/2 NXB MOV 0 N7:34 BND EOR
%   B3:2/0  CNT_SENR_FLT  "FAULT Good Part Sensor Blocked" %
%   B3:6/2  "clear belt" %
%   N7:34  "belt travel since fell part detected" %
% Rung: 9 %
SOR GRT N7:34 N7:29 OTU B3:6/2 EOR
%   N7:34  "belt travel since fell part detected" %
%   N7:29  "belt travel to wipe parts off of belt when fell part detected" %
%   B3:6/2  "clear belt" %
% Rung: 10 %
SOR MOV -256 N10:12 EOR
%   N10:12  "Air Pressure Fault" %
% Rung: 11 %
SOR XIC I:0.1/1 XIC B3:1/4 BST LES N7:25 55 NXB XIC B3:2/7 BND XIO B3:1/14 BST OTE B3:2/7 NXB MOV 255 N10:12 BND EOR
%   I:0.1/1  CRM_ON  "Main Power On" %
%   B3:1/4  "bypass air fault" %
%   N7:25  MAIN_AIR  "converted pressure to psi" %
%   B3:2/7  "Air Pressure Low" %
%   B3:1/14  HMI_RESET_PB  "HMI Fault Reset Pushbutton" %
%   N10:12  "Air Pressure Fault" %
% Rung: 12 %
SOR BST XIC B3:2/6 NXB XIC B3:2/4 BND XIO B3:1/14 OTE B3:2/4 EOR
%   B3:2/6  EDIT  "Edit Required" %
%   B3:2/4  REJECT_RATE_FLT  "FAULT Reject Rate Increased "Parts Flow"" %
%   B3:1/14  HMI_RESET_PB  "HMI Fault Reset Pushbutton" %
% Rung: 13 %
SOR MOV -256 N10:11 EOR
%   N10:11  "Feeder Track Sensor Blocked" %

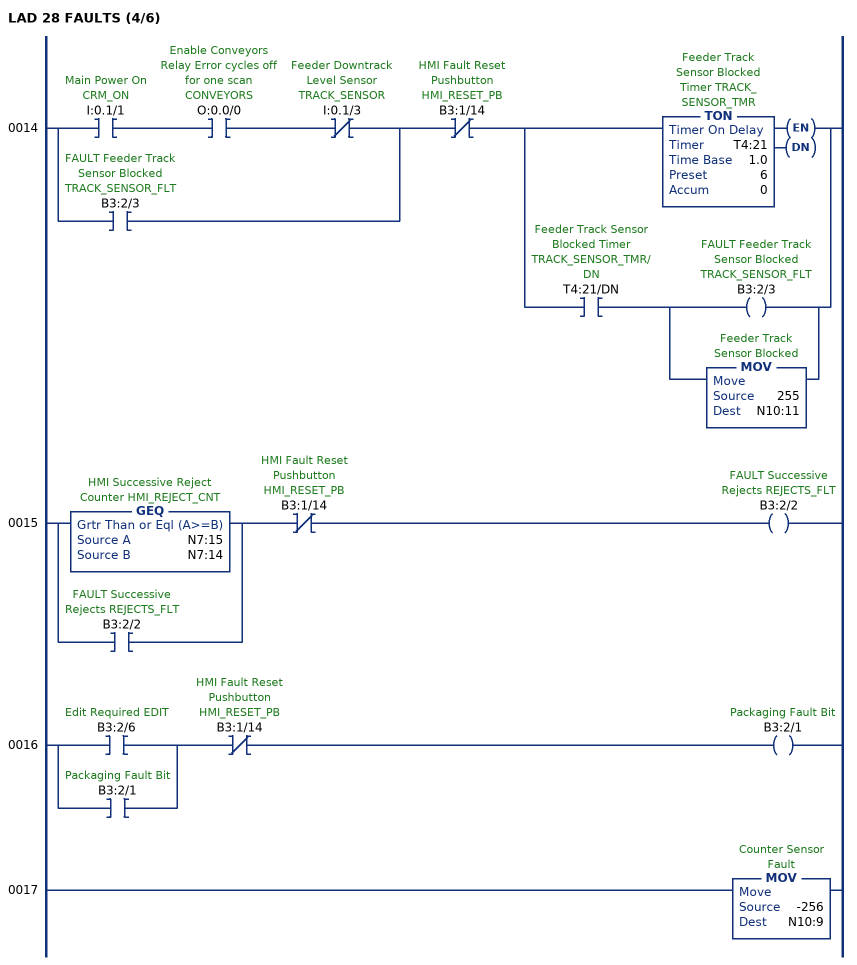
% Rung: 14 %
SOR BST XIC I:0.1/1 XIC O:0.0/0 XIO I:0.1/3 NXB XIC B3:2/3 BND XIO B3:1/14 BST TON T4:21 1.0 6 0 NXB XIC T4:21/DN BST OTE B3:2/3 NXB MOV 255 N10:11 BND BND EOR
%   I:0.1/1  CRM_ON  "Main Power On" %
%   O:0.0/0  CONVEYORS  "Enable Conveyors Relay Error cycles off for one scan" %
%   I:0.1/3  TRACK_SENSOR  "Feeder Downtrack Level Sensor" %
%   B3:2/3  TRACK_SENSOR_FLT  "FAULT Feeder Track Sensor Blocked" %
%   B3:1/14  HMI_RESET_PB  "HMI Fault Reset Pushbutton" %
%   T4:21  TRACK_SENSOR_TMR  "Feeder Track Sensor Blocked Timer" %
%   N10:11  "Feeder Track Sensor Blocked" %
% Rung: 15 %
SOR BST GEQ N7:15 N7:14 NXB XIC B3:2/2 BND XIO B3:1/14 OTE B3:2/2 EOR
%   N7:15  HMI_REJECT_CNT  "HMI Successive Reject Counter" %
%   N7:14  "Succesive Reject Limit" %
%   B3:2/2  REJECTS_FLT  "FAULT Successive Rejects" %
%   B3:1/14  HMI_RESET_PB  "HMI Fault Reset Pushbutton" %
% Rung: 16 %
SOR BST XIC B3:2/6 NXB XIC B3:2/1 BND XIO B3:1/14 OTE B3:2/1 EOR
%   B3:2/6  EDIT  "Edit Required" %
%   B3:2/1  "Packaging Fault Bit" %
%   B3:1/14  HMI_RESET_PB  "HMI Fault Reset Pushbutton" %
% Rung: 17 %
SOR MOV -256 N10:9 EOR
%   N10:9  "Counter Sensor Fault" %

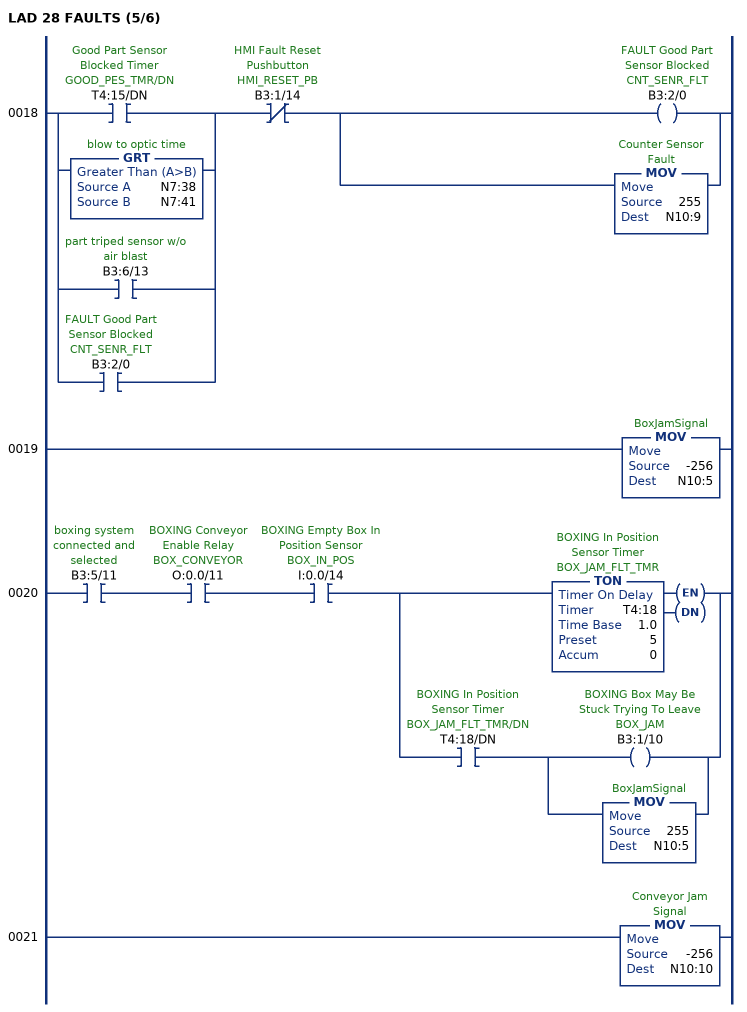
% Rung: 18 %
SOR BST XIC T4:15/DN NXB GRT N7:38 N7:41 NXB XIC B3:6/13 NXB XIC B3:2/0 BND XIO B3:1/14 BST OTE B3:2/0 NXB MOV 255 N10:9 BND EOR
%   T4:15  GOOD_PES_TMR  "Good Part Sensor Blocked Timer" %
%   N7:38  "blow to optic time" %
%   B3:6/13  "part triped sensor w/o air blast" %
%   B3:2/0  CNT_SENR_FLT  "FAULT Good Part Sensor Blocked" %
%   B3:1/14  HMI_RESET_PB  "HMI Fault Reset Pushbutton" %
%   N10:9  "Counter Sensor Fault" %
% Rung: 19 %
SOR MOV -256 N10:5 EOR
%   N10:5  "BoxJamSignal" %
% Rung: 20 %
SOR XIC B3:5/11 XIC O:0.0/11 XIC I:0.0/14 BST TON T4:18 1.0 5 0 NXB XIC T4:18/DN BST OTE B3:1/10 NXB MOV 255 N10:5 BND BND EOR
%   B3:5/11  "boxing system connected and selected" %
%   O:0.0/11  BOX_CONVEYOR  "BOXING Conveyor Enable Relay" %
%   I:0.0/14  BOX_IN_POS  "BOXING Empty Box In Position Sensor" %
%   T4:18  BOX_JAM_FLT_TMR  "BOXING In Position Sensor Timer" %
%   B3:1/10  BOX_JAM  "BOXING Box May Be Stuck Trying To Leave" %
%   N10:5  "BoxJamSignal" %
% Rung: 21 %
SOR MOV -256 N10:10 EOR
%   N10:10  "Conveyor Jam Signal" %

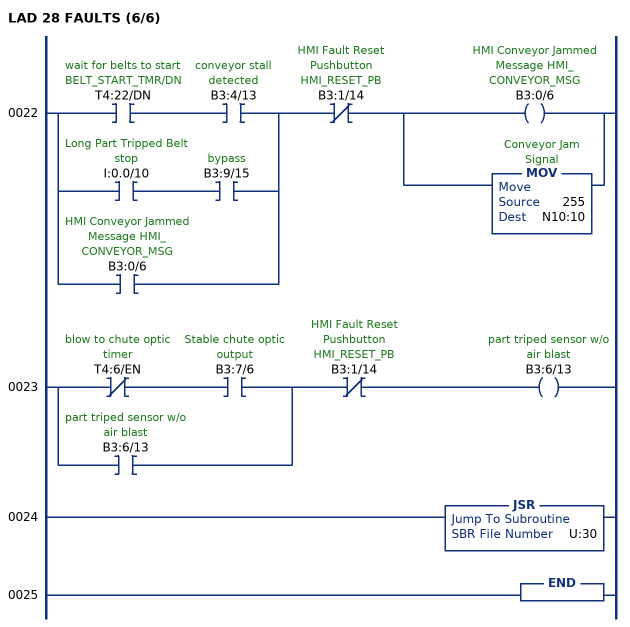
% Rung: 22 %
SOR BST XIC T4:22/DN XIC B3:4/13 NXB XIC I:0.0/10 XIC B3:9/15 NXB XIC B3:0/6 BND XIO B3:1/14 BST OTE B3:0/6 NXB MOV 255 N10:10 BND EOR
%   T4:22  BELT_START_TMR  "wait for belts to start" %
%   B3:4/13  "conveyor stall detected" %
%   I:0.0/10  "Long Part Tripped Belt stop" %
%   B3:9/15  "bypass" %
%   B3:0/6  HMI_CONVEYOR_MSG  "HMI Conveyor Jammed Message" %
%   B3:1/14  HMI_RESET_PB  "HMI Fault Reset Pushbutton" %
%   N10:10  "Conveyor Jam Signal" %
% Rung: 23 %
SOR BST XIO T4:6/EN XIC B3:7/6 NXB XIC B3:6/13 BND XIO B3:1/14 OTE B3:6/13 EOR
%   T4:6  "blow to chute optic timer" %
%   B3:7/6  "Stable chute optic output" %
%   B3:6/13  "part triped sensor w/o air blast" %
%   B3:1/14  HMI_RESET_PB  "HMI Fault Reset Pushbutton" %
% Rung: 24 %
SOR JSR U:30 EOR
% Rung: 25 %
SOR END EOR

LADDER 30 "SPEED"
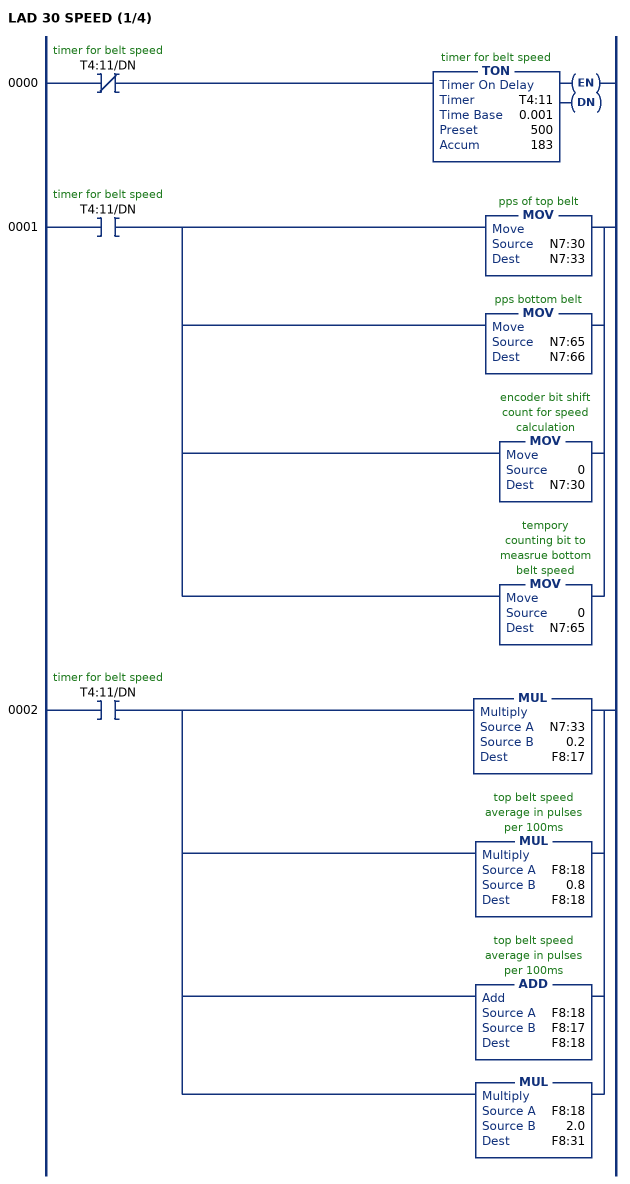
% Rung: 0 %
SOR XIO T4:11/DN TON T4:11 0.001 500 183 EOR
%   T4:11  "timer for belt speed" %
% Rung: 1 %
SOR XIC T4:11/DN BST MOV N7:30 N7:33 NXB MOV N7:65 N7:66 NXB MOV 0 N7:30 NXB MOV 0 N7:65 BND EOR
%   T4:11  "timer for belt speed" %
%   N7:30  "encoder bit shift count for speed calculation" %
%   N7:33  "pps of top belt" %
%   N7:65  "tempory counting bit to measrue bottom belt speed" %
%   N7:66  "pps bottom belt" %
% Rung: 2 %
SOR XIC T4:11/DN BST MUL N7:33 0.2 F8:17 NXB MUL F8:18 0.8 F8:18 NXB ADD F8:18 F8:17 F8:18 NXB MUL F8:18 2.0 F8:31 BND EOR
%   T4:11  "timer for belt speed" %
%   N7:33  "pps of top belt" %
%   F8:18  "top belt speed average in pulses per 100ms" %

